{attribute clr [Container(Layout.Stack)]}
{attribute clr [Group(Layout.Scroll)]}
TYPE CUProcessDataBase EXTENDS TcoCore.TcoStruct :
STRUCT
	{attribute wpf [Container(Layout.Stack)]}
	{attribute wpf [Group(Layout.GroupBox)]}
	Header : CuHeader := (Parent := THISSTRUCT);
END_STRUCT
END_TYPE

(* stored: Version 1.1.0.1
   DUT CUProcessDataBase: Id {5f471120-52ab-4133-bd13-00db205800fd} *)
